FUNCTION_BLOCK MODE_AMS (* AUTO/MANUAL/STOP Mode Control *)
  (* Standard: IEC 61499; ApplicationDomain: Machine Control; Function: Mode Control; Type: AUTO/MANUAL/FAULTED *)
  (* Version 0.1, 2006-07-03, JHC, Holobloc Inc, Changed FAULT to STOP; renamed from MODE_AMF. *)
  (* Version 0.0, 2006-06-26, JHC, Holobloc Inc *)
  (* Compiler header: package fb.rt.mach; *)
  (* Compiler Java Sun JDK 1.5.0 *)
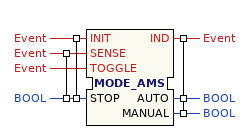
  EVENT_INPUT
    INIT WITH STOP; (* Initialization Request *)
    SENSE WITH STOP;
    TOGGLE; (* Toggle Auto/Manual mode *)
  END_EVENT
  EVENT_OUTPUT
    IND WITH AUTO, MANUAL; (* Mode change indication *)
  END_EVENT
  VAR_INPUT
    STOP : BOOL; (* STOP condition, e.g., FAULT sensor or STOP pushbutton *)
  END_VAR
  VAR_OUTPUT
    AUTO : BOOL;
    MANUAL : BOOL;
  END_VAR
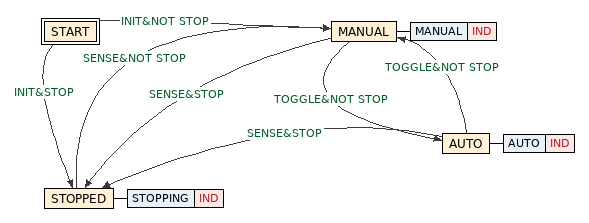
  EC_STATES
    START; (* Initial State *)
    MANUAL : MANUAL -> IND;
    STOPPED : STOPPING -> IND;
    AUTO : AUTO -> IND;
  END_STATES
  EC_TRANSITIONS
    START TO MANUAL := INIT&NOT STOP;
    START TO STOPPED := INIT&STOP;
    MANUAL TO STOPPED := SENSE&STOP;
    AUTO TO STOPPED := SENSE&STOP;
    STOPPED TO MANUAL := SENSE&NOT STOP;
    MANUAL TO AUTO := TOGGLE&NOT STOP;
    AUTO TO MANUAL := TOGGLE&NOT STOP;
  END_TRANSITIONS
  ALGORITHM MANUAL IN ST:
AUTO := FALSE;
MANUAL := TRUE;
  END_ALGORITHM
  ALGORITHM STOPPING IN ST:
AUTO := FALSE;
MANUAL := FALSE;
  END_ALGORITHM
  ALGORITHM AUTO IN ST:
AUTO := TRUE;
MANUAL := FALSE;
  END_ALGORITHM
END_FUNCTION_BLOCK
